{attribute addProperty BoxType "AMI8000-0000-0016"}
{attribute addProperty Id "Target_positionAT %Q*UDINT324"}
{attribute addProperty CRC "1093881770"}
{attribute addProperty SizeInBites "32"}
{attribute addProperty SizeInBytes "4"}
TYPE DRV_Target_position_41334FAA :
STRUCT
	{attribute addProperty Name "Target_position"}
	Target_position AT %Q* : UDINT;
END_STRUCT
END_TYPE

(* stored: Version 1.2.0.0, ProductVersion 3.1.4024.9
   DUT DRV_Target_position_41334FAA: Id {555f2803-7659-41ca-be3c-4bcb9f3ed77d} *)
